PROGRAM PRG_Test
VAR
	validateFunctionsTest : ValidateFunctionsTest;
	manipulateFunctionsTest : ManipulateFunctionsTest;
	convertFunctionsTest : ConvertFunctionsTest;
	
	sb255Test : StringBuilder255Test;
	buildStringInlineTest : BuildStringInlineTest;
	sbExtBufferTest : StringBuilderExtBufferTest;
	sbInfiniteTest : StringBuilderInfiniteTest;
END_VAR

TcUnit.RUN();

END_PROGRAM

(* stored: Version 1.1.0.1, ProductVersion 3.1.4024.15
   POU PRG_Test: Id {f561285f-0a78-0d21-2985-5942483404f0}, SpecialFunc None *)
